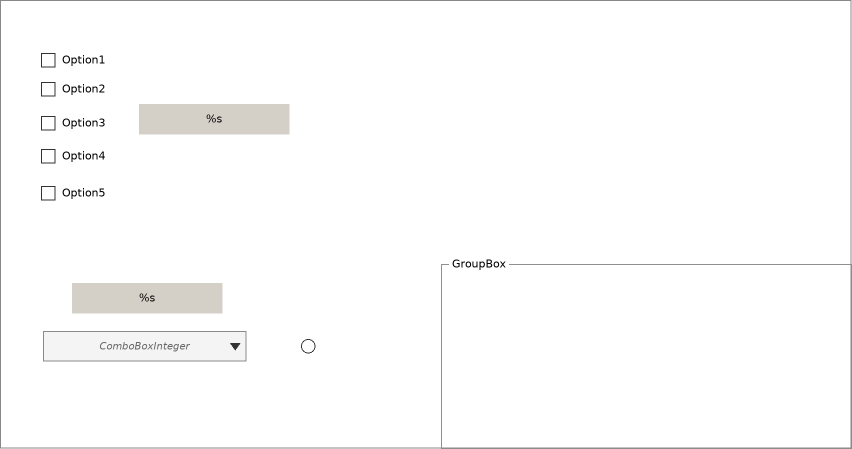
VISUALIZATION P03_Common  // 852x449
    Checkbox (39,45 150x30), "Option1", variable: Main.bCheckBox1
    Checkbox (39,74 150x30), "Option2", variable: Main.bCheckBox2
    Checkbox (39,108 150x30), "Option3", variable: Main.bCheckBox3
    Checkbox (39,141 150x30), "Option4", variable: Main.bCheckBox4
    Checkbox (39,178 150x30), "Option5", variable: Main.bCheckBox5
    Textfield (139,104 150x30), "%s", text variable: Main.sOutput2
    ComboBoxInteger (43,331 203x30), variable: Main.iCombINdex, text list: 'TextList'
    RadioButton (299,271 150x150), variable: Main.iCombINdex
        Areas[0]: Text=Option1
        Areas[1]: Text=Option2
        Areas[2]: Text=Option3
        Areas[3]: Text=Option4
        Areas[4]: Text=Option5
    Textfield (72,283 150x30), "%s", text variable: Main.sOutput
    GroupBox (441,256 411x193), "GroupBox"
END_VISUALIZATION

(* stored: Version 1.1.0.1, ProductVersion 3.1.4024.6
   Visu P03_Common: Id {2365058f-47a6-4ad4-b6fb-409d7c4b596b} *)
